// TIA Portal V16 export
// export: Created 2023-03-29T11:03:47.1842828Z, ExportSetting WithDefaults, DisplayName Totally Integrated Automation Portal, DisplayVersion V16 Update 6, DisplayName TIA Portal Version Control Interface, DisplayVersion V16 Update 2, DisplayName TIA Portal Openness, DisplayVersion V16 Update 6, DisplayName STEP 7 Professional, DisplayVersion V16 Update 6, DisplayName STEP 7 Safety, DisplayVersion V16, DisplayName WinCC Advanced, DisplayVersion V16 Update 6
VAR_GLOBAL   // PLC tag table "Tag Sim"
   Sim_23 AT %M3002.6 : Bool;
   Sim_22 AT %M3002.5 : Bool;
   Sim_21 AT %M3002.4 : Bool;
   Sim_24 AT %M3002.7 : Bool;
   Sim_19 AT %M3002.2 : Bool;
   Sim_generator_reg AT %M3002.3 : Bool;
   Sim__Z5_Open_Spust AT %M3001.1 : Bool;
   Sim__Z2_Colse_Wlot AT %M3000.2 : Bool;
   Sim__Z6_Open_Wlot AT %M3001.3 : Bool;
   Sim__Z1_Open_Spust AT %M3000.1 : Bool;
   Sim__Z1_Close_Spust AT %M3000.0 : Bool;
   Sim__Z6_Close_Wlot AT %M3001.2 : Bool;
   Sim__Z8_Close_Wylot AT %M3001.6 : Bool;
   Sim__Z3_Open_Spust AT %M3000.5 : Bool;
   Sim__Z9_Close AT %M3002.0 : Bool;
   Sim__Z5_Close_Spust AT %M3001.0 : Bool;
   Sim__Z3_Close_Spust AT %M3000.4 : Bool;
   Sim__Z4_Close_Wlot AT %M3000.6 : Bool;
   Sim__Z2_Open_Wlot AT %M3000.3 : Bool;
   Sim__Z9_Open AT %M3002.1 : Bool;
   Sim__Z8_Open_Wlot AT %M3001.7 : Bool;
   Sim__Z4_Open_Wlot AT %M3000.7 : Bool;
   Sim__Z7_Close_Spust AT %M3001.4 : Bool;
   Sim__Z7_Open_Spust AT %M3001.5 : Bool;
   Sim__Z7_TCP_error AT %M3003.0 : Bool;
   Sim__Z10_close AT %M3003.2 : Bool;
   Sim__Z10_open AT %M3003.1 : Bool;
   "auto set open" AT %M3003.3 : Bool;
   "auto set close" AT %M3003.4 : Bool;
END_VAR
